PROGRAM MAIN
VAR
	fbFilterWheel : FB_XTESFilterWheel;
	bExecute: BOOL;
	sTestCmd: STRING;
	nSetPos: USINT;
	nGetPos: USINT;
	bBusy: BOOL;
	sTestResponse: STRING;
	sError: STRING;
END_VAR

fbFilterWheel(bExecute:=bExecute,
	sTestCmd:=sTestCmd,
	stIn_EL6001:=GVL.stIn_EL6001,
	stOut_EL6001:=GVL.stOut_EL6001,
	nSetPos:=nSetPos,
	nGetPos=>nGetPos,
	bBusy=>bBusy,
	bError=>,
	sError=>sError,
	sTestResponse=>sTestResponse);

END_PROGRAM

(* stored: Version 1.1.0.1, ProductVersion 3.1.4020.14
   POU MAIN: Id {1e57a20e-abc8-4724-b740-d22e8c3d8d13}, SpecialFunc None *)
